(* PLC project mtcs, Institute of Astronomy OntoManager 0.0.1 *)
(* stored: creationDateTime 2017-02-07T02:01:16.949163, modificationDateTime 2017-02-07T02:01:16.949163 *)

TYPE MTCSParts : STRUCT
  telemetry : Telemetry;  (* The telemetry *)
  cover : Cover;  (* The Cover of the telescope *)
  m1 : M1;  (* The primary mirror of the telescope *)
  m2 : M2;  (* The secondary mirror of the telescope *)
  m3 : M3;  (* The tertiary mirror of the telescope *)
  services : Services;  (* The Services system *)
  safety : Safety;  (* The safety *)
  hydraulics : Hydraulics;  (* The hydraulics *)
  axes : Axes;  (* The axes *)
  dome : Dome;  (* The dome *)
  configManager : ConfigManager;  (* The config manager (to load/save/activate configuration data) *)
END_STRUCT;
END_TYPE

TYPE MTCSProcesses : STRUCT
  initialize : Process;  (* Start initializing the whole MTCS *)
  lock : Process;  (* Lock the whole MTCS *)
  unlock : Process;  (* Unlock the whole MTCS *)
  changeOperator : ChangeOperatorStateProcess;  (* Change the operator (e.g. OBSERVER, TECH, ...) *)
  verifyPassword : ChangeOperatorStateProcess;  (* Only verify the operator password *)
  reboot : Process;  (* Reboot the whole MTCS *)
  shutdown : Process;  (* Shutdown the whole MTCS *)
  wakeUp : Process;  (* Wake up the whole MTCS *)
  goToSleep : Process;  (* Let the whole MTCS go to sleep *)
  stop : Process;  (* Stop the dome and telescope *)
  endOfNight : Process;  (* End of night *)
  changeInstrument : MTCSChangeInstrumentProcess;  (* Change the instrument *)
  park : MTCSParkProcess;  (* Park the telescope (including Axes, Dome, M3, ...) *)
  point : MTCSPointProcess;  (* Point the telescope and dome to a new target *)
END_STRUCT;
END_TYPE

TYPE MTCSStatuses : STRUCT
  initializationStatus : InitializationStatus;
  healthStatus : HealthStatus;
  busyStatus : BusyStatus;
  operatorStatus : OperatorStatus;
  passwordHealthStatus : HealthStatus;
  activityStatus : ActivityStatus;
END_STRUCT;
END_TYPE

TYPE MTCSInstrumentsConfig : STRUCT
  instrument0 : InstrumentConfig;  (* Instrument 0 *)
  instrument1 : InstrumentConfig;  (* Instrument 1 *)
  instrument2 : InstrumentConfig;  (* Instrument 2 *)
  instrument3 : InstrumentConfig;  (* Instrument 3 *)
  instrument4 : InstrumentConfig;  (* Instrument 4 *)
  instrument5 : InstrumentConfig;  (* Instrument 5 *)
  instrument6 : InstrumentConfig;  (* Instrument 6 *)
  instrument7 : InstrumentConfig;  (* Instrument 7 *)
  instrument8 : InstrumentConfig;  (* Instrument 8 *)
  instrument9 : InstrumentConfig;  (* Instrument 9 *)
END_STRUCT;
END_TYPE

TYPE MTCSParkPositionConfig : STRUCT
  name : STRING;  (* The name of the position (e.g. 'PARK') *)
  axes : STRING;  (* Name of the corresponding Axes position *)
  doAxes : BOOL;  (* Change the Axes to the 'axes' position *)
  m3 : STRING;  (* Name of the corresponding M3 position *)
  doM3 : BOOL;  (* Change M3 to the 'm3' position *)
  dome : STRING;  (* Name of the corresponding dome position *)
  doDome : BOOL;  (* Change M3 to the 'm3' position *)
END_STRUCT;
END_TYPE

TYPE MTCSParkPositionsConfig : STRUCT
  position0 : MTCSParkPositionConfig;  (* Park position 0 *)
  position1 : MTCSParkPositionConfig;  (* Park position 1 *)
  position2 : MTCSParkPositionConfig;  (* Park position 2 *)
  position3 : MTCSParkPositionConfig;  (* Park position 3 *)
  position4 : MTCSParkPositionConfig;  (* Park position 4 *)
  position5 : MTCSParkPositionConfig;  (* Park position 5 *)
  position6 : MTCSParkPositionConfig;  (* Park position 6 *)
  position7 : MTCSParkPositionConfig;  (* Park position 7 *)
  position8 : MTCSParkPositionConfig;  (* Park position 8 *)
  position9 : MTCSParkPositionConfig;  (* Park position 9 *)
END_STRUCT;
END_TYPE

TYPE MTCSEndOfNightStepConfig : STRUCT
  parkAxes : BOOL;  (* Park the telescope *)
  parkAxesPosition : STRING;  (* Position to park the telescope *)
  parkTelescopeWait : BOOL;  (* Wait until the telescope is parked *)
  parkM3 : BOOL;  (* Park M3 *)
  parkM3Position : STRING;  (* Position to park M3 *)
  parkM3Wait : BOOL;  (* Wait until M3 is parked *)
  parkDome : BOOL;  (* Park the dome *)
  parkDomePosition : STRING;  (* Position to park the dome *)
  parkDomeWait : BOOL;  (* Wait until the dome is parked *)
  closeCover : BOOL;  (* Close the cover *)
  closeCoverWait : BOOL;  (* Wait until the cover is closed *)
  closeDome : BOOL;  (* Close the dome *)
  closeDomeWait : BOOL;  (* Wait until the dome is closed *)
  stop : BOOL;  (* Stop the axes and dome *)
  stopWait : BOOL;  (* Wait until the axes and dome are stopped *)
  goToSleep : BOOL;  (* Make the telescope go to sleep *)
  goToSleepWait : BOOL;  (* Wait until the telescope is sleeping *)
END_STRUCT;
END_TYPE

TYPE MTCSEndOfNightConfig : STRUCT
  step0 : MTCSEndOfNightStepConfig;  (* Step 0 *)
  step1 : MTCSEndOfNightStepConfig;  (* Step 1 *)
  step2 : MTCSEndOfNightStepConfig;  (* Step 2 *)
  step3 : MTCSEndOfNightStepConfig;  (* Step 3 *)
  step4 : MTCSEndOfNightStepConfig;  (* Step 4 *)
  step5 : MTCSEndOfNightStepConfig;  (* Step 5 *)
  step6 : MTCSEndOfNightStepConfig;  (* Step 6 *)
  step7 : MTCSEndOfNightStepConfig;  (* Step 7 *)
  step8 : MTCSEndOfNightStepConfig;  (* Step 8 *)
  step9 : MTCSEndOfNightStepConfig;  (* Step 9 *)
  step10 : MTCSEndOfNightStepConfig;  (* Step 10 *)
  step11 : MTCSEndOfNightStepConfig;  (* Step 11 *)
  step12 : MTCSEndOfNightStepConfig;  (* Step 12 *)
  step13 : MTCSEndOfNightStepConfig;  (* Step 13 *)
  step14 : MTCSEndOfNightStepConfig;  (* Step 14 *)
  step15 : MTCSEndOfNightStepConfig;  (* Step 15 *)
  step16 : MTCSEndOfNightStepConfig;  (* Step 16 *)
  step17 : MTCSEndOfNightStepConfig;  (* Step 17 *)
  step18 : MTCSEndOfNightStepConfig;  (* Step 18 *)
  step19 : MTCSEndOfNightStepConfig;  (* Step 19 *)
END_STRUCT;
END_TYPE

TYPE MTCSConfig : STRUCT
  instruments : MTCSInstrumentsConfig;  (* Configure the instruments *)
  endOfNight : MTCSEndOfNightConfig;  (* Configure the instruments *)
  parkPositions : MTCSParkPositionsConfig;  (* Configure the park positions of the telescope (dome+telescope+m3+...) *)
END_STRUCT;
END_TYPE

TYPE MTCSChangeInstrumentProcessArgs : STRUCT
  name : STRING;  (* Name of the instrument *)
END_STRUCT;
END_TYPE

TYPE MTCSParkProcessArgs : STRUCT
  name : STRING;  (* Name of the park position *)
END_STRUCT;
END_TYPE

TYPE MTCSPointProcessArgs : STRUCT
  alphaUnits : AxesAlphaUnits;  (* The units in which alpha is given *)
  alpha : LREAL;  (* Right ascention, in the units of the alphaUnits argument *)
  deltaUnits : AxesDeltaUnits;  (* The units in which delta is given *)
  delta : LREAL;  (* Declination, in the units of the deltaUnits argument *)
  muUnits : AxesMuUnits;  (* The units in which muAlpha and muDelta are given *)
  muAlpha : LREAL;  (* Right ascention proper motion, the units of muUmits (do not multiply by cos(delta)!) *)
  muDelta : LREAL;  (* Declination proper motion, in radians/year *)
  parallax : LREAL;  (* Object parallax, in arcseconds *)
  radialVelocity : LREAL;  (* Object radial velocity, in km/s *)
  epoch : LREAL := 2000;  (* Epoch, e.g. 2000.0 *)
  tracking : BOOL := TRUE;  (* True to start tracking the object, false to Only do a pointing *)
  rotUnits : AxesMoveUnits;  (* Units of the 'rot', 'roc' and 'ron' arguments (RADIANS, DEGREES, ARCSECONDS, ...) *)
  rotOffset : LREAL;  (* Offset to move the currently active rotator (incompatible with 'roc' and 'ron' args) *)
  rocOffset : LREAL;  (* Offset to move the cassegrain rotation axis (incompatible with 'rot' arg) *)
  ronOffset : LREAL;  (* Offset to move the nasmyth rotation axis (incompatible with 'rot' arg) *)
  doRotOffset : BOOL;  (* True to move the currently active rotator, false to leave it untouched *)
  doRocOffset : BOOL;  (* True to move the cassegrain rotation axis, false to leave it untouched *)
  doRonOffset : BOOL;  (* True to move the nasmyth rotation axis, false to leave it untouched *)
  doDomeTracking : BOOL := TRUE;  (* True to enable dome tracking *)
END_STRUCT;
END_TYPE

FUNCTION_BLOCK SM_MTCS
  VAR_INPUT
    {attribute 'OPC.UA.DA' := '1'}
    {attribute 'OPC.UA.DA.Access' := '1'}
    editableConfig : MTCSConfig;  (* Editable configuration of the MTCS *)
  END_VAR
  VAR_OUTPUT
    {attribute 'OPC.UA.DA' := '1'}
    {attribute 'OPC.UA.DA.Access' := '1'}
    actualStatus : STRING;  (* Current status description *)
    previousStatus : STRING;  (* Previous status description *)
    {attribute 'OPC.UA.DA' := '1'}
    {attribute 'OPC.UA.DA.Access' := '1'}
    noOfFailedOperatorChanges : UINT;  (* How many times has a wrong password been entered? *)
    {attribute 'OPC.UA.DA' := '1'}
    {attribute 'OPC.UA.DA.Access' := '1'}
    activeInstrument : InstrumentConfig;  (* Config of the currently active instrument (depending on M3 and possibly derotator) *if* isInstrumentActive is TRUE *)
    {attribute 'OPC.UA.DA' := '1'}
    {attribute 'OPC.UA.DA.Access' := '1'}
    activeInstrumentNumber : INT;  (* Number of the currently active instrument (0..9, or -1 if no instrument is active) *)
    {attribute 'OPC.UA.DA' := '1'}
    {attribute 'OPC.UA.DA.Access' := '1'}
    activeInstrumentName : STRING;  (* Name of the currently active instrument *)
    {attribute 'OPC.UA.DA' := '1'}
    {attribute 'OPC.UA.DA.Access' := '1'}
    isInstrumentActive : BOOL;  (* Is an instrument currently active (i.e. is M3 static at a known position?) *)
    {attribute 'OPC.UA.DA' := '1'}
    {attribute 'OPC.UA.DA.Access' := '1'}
    config : MTCSConfig;  (* Active configuration of the ServicesTiming subsystem *)
    statuses : MTCSStatuses;  (* Statuses of the state machine *)
    parts : MTCSParts;  (* Parts of the state machine *)
    processes : MTCSProcesses;  (* Processes of the state machine *)
  END_VAR

            parts.telemetry( operatorStatus := statuses.operatorStatus );
parts.cover(
    operatorStatus := statuses.operatorStatus,
    aziPos := parts.axes.parts.azi.actPos,
    elePos := parts.axes.parts.ele.actPos);
parts.m1(
    operatorStatus := statuses.operatorStatus,
    tubeAngleMeasurement := parts.telemetry.parts.accelerometers.tube);
parts.m2(
    operatorStatus := statuses.operatorStatus,
    io := parts.m1.parts.io,
    actualFocalStation := parts.m3.actualKnownPositionID,
    m3KnownPositionsConfig := parts.m3.config.knownPositions,
    temperatures := parts.telemetry.parts.temperatures);
parts.m3( operatorStatus := statuses.operatorStatus );
parts.services( operatorStatus := statuses.operatorStatus );
parts.safety(
    operatorStatus := statuses.operatorStatus,
    activityStatus := statuses.activityStatus);
parts.hydraulics(
    operatorStatus := statuses.operatorStatus,
    safetyHydraulics := parts.safety.parts.hydraulics,
    safetyIO := parts.safety.parts.io);
parts.dome(
    operatorStatus := statuses.operatorStatus,
    aziPos := parts.axes.parts.azi.actPos);
parts.configManager( isEnabled := statuses.operatorStatus.tech );
statuses.initializationStatus();
statuses.healthStatus(
    isGood := parts.axes.statuses.healthStatus.isGood AND (parts.cover.statuses.healthStatus.isGood AND (parts.m1.statuses.healthStatus.isGood AND (parts.m2.statuses.healthStatus.isGood AND (parts.m3.statuses.healthStatus.isGood AND (parts.services.statuses.healthStatus.isGood AND (parts.telemetry.statuses.healthStatus.isGood AND (parts.safety.statuses.healthStatus.isGood AND (parts.hydraulics.statuses.healthStatus.isGood AND parts.dome.statuses.healthStatus.isGood)))))))),
    hasWarning := parts.axes.statuses.healthStatus.hasWarning OR (parts.cover.statuses.healthStatus.hasWarning OR (parts.m1.statuses.healthStatus.hasWarning OR (parts.m2.statuses.healthStatus.hasWarning OR (parts.m3.statuses.healthStatus.hasWarning OR (parts.services.statuses.healthStatus.hasWarning OR (parts.telemetry.statuses.healthStatus.hasWarning OR (parts.safety.statuses.healthStatus.hasWarning OR (parts.hydraulics.statuses.healthStatus.hasWarning OR parts.dome.statuses.healthStatus.hasWarning)))))))));
statuses.busyStatus( isBusy := parts.axes.statuses.busyStatus.busy OR (parts.cover.statuses.busyStatus.busy OR (parts.m1.statuses.busyStatus.busy OR (parts.m2.statuses.busyStatus.busy OR (parts.m3.statuses.busyStatus.busy OR (parts.services.statuses.busyStatus.busy OR (parts.telemetry.statuses.busyStatus.busy OR (parts.safety.statuses.busyStatus.busy OR (parts.hydraulics.statuses.busyStatus.busy OR parts.dome.statuses.busyStatus.busy)))))))) );
statuses.operatorStatus();
statuses.passwordHealthStatus( superState := statuses.operatorStatus.observer );
statuses.activityStatus(
    superState := statuses.initializationStatus.initialized OR statuses.initializationStatus.initializingFailed,
    isAwake := (parts.hydraulics.pumpsState = HydraulicsPumpsStates.RUNNING) OR parts.axes.statuses.poweredStatus.enabled,
    isMoving := parts.axes.statuses.busyStatus.busy OR parts.axes.isTracking);
processes.initialize( isEnabled := NOT(statuses.initializationStatus.initializing) );
processes.lock( isEnabled := statuses.operatorStatus.tech AND statuses.initializationStatus.initialized );
processes.unlock( isEnabled := statuses.operatorStatus.tech AND statuses.initializationStatus.locked );
processes.changeOperator( isEnabled := TRUE );
processes.verifyPassword( isEnabled := TRUE );
processes.reboot( isEnabled := TRUE );
processes.shutdown( isEnabled := statuses.operatorStatus.tech );
processes.wakeUp( isEnabled := statuses.activityStatus.sleeping );
processes.goToSleep( isEnabled := statuses.activityStatus.awake OR statuses.healthStatus.bad );
processes.stop( isEnabled := statuses.initializationStatus.initialized );
processes.endOfNight( isEnabled := TRUE );
processes.changeInstrument( isEnabled := statuses.initializationStatus.initialized OR statuses.healthStatus.bad );
processes.park( isEnabled := parts.axes.statuses.busyStatus.idle AND (parts.dome.statuses.busyStatus.idle AND parts.m3.statuses.busyStatus.idle) );
processes.point( isEnabled := parts.axes.processes.point.statuses.enabledStatus.enabled AND parts.dome.processes.trackAxes.statuses.enabledStatus.enabled );

          

{attribute 'TcRpcEnable' := '1'}
METHOD initialize : RequestResults
                  initialize := THIS^.processes.initialize.request();

                
END_METHOD

{attribute 'TcRpcEnable' := '1'}
METHOD lock : RequestResults
                  lock := THIS^.processes.lock.request();

                
END_METHOD

{attribute 'TcRpcEnable' := '1'}
METHOD unlock : RequestResults
                  unlock := THIS^.processes.unlock.request();

                
END_METHOD

{attribute 'TcRpcEnable' := '1'}
METHOD changeOperator : RequestResults
  VAR_INPUT
    state : OperatorStates;
    password : STRING;
  END_VAR
                  changeOperator := THIS^.processes.changeOperator.request(
    state := state,
    password := password);

                
END_METHOD

{attribute 'TcRpcEnable' := '1'}
METHOD verifyPassword : RequestResults
  VAR_INPUT
    state : OperatorStates;
    password : STRING;
  END_VAR
                  verifyPassword := THIS^.processes.verifyPassword.request(
    state := state,
    password := password);

                
END_METHOD

{attribute 'TcRpcEnable' := '1'}
METHOD reboot : RequestResults
                  reboot := THIS^.processes.reboot.request();

                
END_METHOD

{attribute 'TcRpcEnable' := '1'}
METHOD shutdown : RequestResults
                  shutdown := THIS^.processes.shutdown.request();

                
END_METHOD

{attribute 'TcRpcEnable' := '1'}
METHOD wakeUp : RequestResults
                  wakeUp := THIS^.processes.wakeUp.request();

                
END_METHOD

{attribute 'TcRpcEnable' := '1'}
METHOD goToSleep : RequestResults
                  goToSleep := THIS^.processes.goToSleep.request();

                
END_METHOD

{attribute 'TcRpcEnable' := '1'}
METHOD stop : RequestResults
                  stop := THIS^.processes.stop.request();

                
END_METHOD

{attribute 'TcRpcEnable' := '1'}
METHOD endOfNight : RequestResults
                  endOfNight := THIS^.processes.endOfNight.request();

                
END_METHOD

{attribute 'TcRpcEnable' := '1'}
METHOD changeInstrument : RequestResults
  VAR_INPUT
    name : STRING;
  END_VAR
                  changeInstrument := THIS^.processes.changeInstrument.request( name := name );

                
END_METHOD

{attribute 'TcRpcEnable' := '1'}
METHOD park : RequestResults
  VAR_INPUT
    name : STRING;
  END_VAR
                  park := THIS^.processes.park.request( name := name );

                
END_METHOD

{attribute 'TcRpcEnable' := '1'}
METHOD point : RequestResults
  VAR_INPUT
    alphaUnits : AxesAlphaUnits;
    alpha : LREAL;
    deltaUnits : AxesDeltaUnits;
    delta : LREAL;
    muUnits : AxesMuUnits;
    muAlpha : LREAL;
    muDelta : LREAL;
    parallax : LREAL;
    radialVelocity : LREAL;
    epoch : LREAL;
    tracking : BOOL;
    rotUnits : AxesMoveUnits;
    rotOffset : LREAL;
    rocOffset : LREAL;
    ronOffset : LREAL;
    doRotOffset : BOOL;
    doRocOffset : BOOL;
    doRonOffset : BOOL;
    doDomeTracking : BOOL;
  END_VAR
                  point := THIS^.processes.point.request(
    alphaUnits := alphaUnits,
    alpha := alpha,
    deltaUnits := deltaUnits,
    delta := delta,
    muUnits := muUnits,
    muAlpha := muAlpha,
    muDelta := muDelta,
    parallax := parallax,
    radialVelocity := radialVelocity,
    epoch := epoch,
    tracking := tracking,
    rotUnits := rotUnits,
    rotOffset := rotOffset,
    rocOffset := rocOffset,
    ronOffset := ronOffset,
    doRotOffset := doRotOffset,
    doRocOffset := doRocOffset,
    doRonOffset := doRonOffset,
    doDomeTracking := doDomeTracking);

                
END_METHOD

{attribute 'TcRpcEnable' := '1'}
METHOD _log : BOOL
  VAR_INPUT
    name : STRING;  (* Name of this function block instance *)
  END_VAR
  VAR_IN_OUT
    buffer : LogBuffer;  (* Buffer to write all logging to *)
  END_VAR
  VAR
    subBuffer : LogBuffer;  (* Temporary buffer to write logging by parts (sub-statemachines) to *)
  END_VAR
                  THIS^.parts.telemetry._log(
    name := 'telemetry',
    buffer := subBuffer);
THIS^.parts.cover._log(
    name := 'cover',
    buffer := subBuffer);
THIS^.parts.m1._log(
    name := 'm1',
    buffer := subBuffer);
THIS^.parts.m2._log(
    name := 'm2',
    buffer := subBuffer);
THIS^.parts.m3._log(
    name := 'm3',
    buffer := subBuffer);
THIS^.parts.services._log(
    name := 'services',
    buffer := subBuffer);
THIS^.parts.safety._log(
    name := 'safety',
    buffer := subBuffer);
THIS^.parts.hydraulics._log(
    name := 'hydraulics',
    buffer := subBuffer);
THIS^.parts.axes._log(
    name := 'axes',
    buffer := subBuffer);
THIS^.parts.dome._log(
    name := 'dome',
    buffer := subBuffer);
THIS^.parts.configManager._log(
    name := 'configManager',
    buffer := subBuffer);
LOGGER(
    name := name,
    actualStatus := THIS^.actualStatus,
    previousStatus := THIS^.previousStatus,
    buffer := buffer,
    subBuffer := subBuffer,
    pHealthStatus := ADR(THIS^.statuses.healthStatus),
    pBusyStatus := ADR(THIS^.statuses.busyStatus));

                
END_METHOD
END_FUNCTION_BLOCK

FUNCTION_BLOCK MTCSChangeInstrumentProcess EXTENDS BaseProcess
  VAR_INPUT
    {attribute 'OPC.UA.DA' := '1'}
    set : MTCSChangeInstrumentProcessArgs;  (* Arguments to be set, before writing do_request TRUE *)
  END_VAR
  VAR_OUTPUT
    {attribute 'OPC.UA.DA' := '1'}
    {attribute 'OPC.UA.DA.Access' := '1'}
    get : MTCSChangeInstrumentProcessArgs;  (* Arguments in use by the process, if do_request was accepted *)
  END_VAR

            IF do_request THEN
    do_request_result := request( name := set.name );
    do_request := FALSE;
END_IF;
SUPER^();

          

{attribute 'TcRpcEnable' := '1'}
METHOD start
  VAR_INPUT
    name : STRING;  (* Name of the instrument *)
  END_VAR
                  THIS^.get.name := name;
THIS^.statuses.busyStatus( isBusy := TRUE );
THIS^.statuses.healthStatus( isGood := TRUE );

                
END_METHOD

{attribute 'TcRpcEnable' := '1'}
METHOD request : RequestResults
  VAR_INPUT
    name : STRING;  (* Name of the instrument *)
  END_VAR
                  IF THIS^.statuses.enabledStatus.enabled THEN
    THIS^.start( name := name );
    request := RequestResults.ACCEPTED;
ELSE
    request := RequestResults.REJECTED;
END_IF;

                
END_METHOD
END_FUNCTION_BLOCK

FUNCTION_BLOCK MTCSParkProcess EXTENDS BaseProcess
  VAR_INPUT
    {attribute 'OPC.UA.DA' := '1'}
    set : MTCSParkProcessArgs;  (* Arguments to be set, before writing do_request TRUE *)
  END_VAR
  VAR_OUTPUT
    {attribute 'OPC.UA.DA' := '1'}
    {attribute 'OPC.UA.DA.Access' := '1'}
    get : MTCSParkProcessArgs;  (* Arguments in use by the process, if do_request was accepted *)
  END_VAR

            IF do_request THEN
    do_request_result := request( name := set.name );
    do_request := FALSE;
END_IF;
SUPER^();

          

{attribute 'TcRpcEnable' := '1'}
METHOD start
  VAR_INPUT
    name : STRING;  (* Name of the park position *)
  END_VAR
                  THIS^.get.name := name;
THIS^.statuses.busyStatus( isBusy := TRUE );
THIS^.statuses.healthStatus( isGood := TRUE );

                
END_METHOD

{attribute 'TcRpcEnable' := '1'}
METHOD request : RequestResults
  VAR_INPUT
    name : STRING;  (* Name of the park position *)
  END_VAR
                  IF THIS^.statuses.enabledStatus.enabled THEN
    THIS^.start( name := name );
    request := RequestResults.ACCEPTED;
ELSE
    request := RequestResults.REJECTED;
END_IF;

                
END_METHOD
END_FUNCTION_BLOCK

FUNCTION_BLOCK MTCSPointProcess EXTENDS BaseProcess
  VAR_INPUT
    {attribute 'OPC.UA.DA' := '1'}
    set : MTCSPointProcessArgs;  (* Arguments to be set, before writing do_request TRUE *)
  END_VAR
  VAR_OUTPUT
    {attribute 'OPC.UA.DA' := '1'}
    {attribute 'OPC.UA.DA.Access' := '1'}
    get : MTCSPointProcessArgs;  (* Arguments in use by the process, if do_request was accepted *)
  END_VAR

            IF do_request THEN
    do_request_result := request(
    alphaUnits := set.alphaUnits,
    alpha := set.alpha,
    deltaUnits := set.deltaUnits,
    delta := set.delta,
    muUnits := set.muUnits,
    muAlpha := set.muAlpha,
    muDelta := set.muDelta,
    parallax := set.parallax,
    radialVelocity := set.radialVelocity,
    epoch := set.epoch,
    tracking := set.tracking,
    rotUnits := set.rotUnits,
    rotOffset := set.rotOffset,
    rocOffset := set.rocOffset,
    ronOffset := set.ronOffset,
    doRotOffset := set.doRotOffset,
    doRocOffset := set.doRocOffset,
    doRonOffset := set.doRonOffset,
    doDomeTracking := set.doDomeTracking);
    do_request := FALSE;
END_IF;
SUPER^();

          

{attribute 'TcRpcEnable' := '1'}
METHOD start
  VAR_INPUT
    alphaUnits : AxesAlphaUnits;  (* The units in which alpha is given *)
    alpha : LREAL;  (* Right ascention, in the units of the alphaUnits argument *)
    deltaUnits : AxesDeltaUnits;  (* The units in which delta is given *)
    delta : LREAL;  (* Declination, in the units of the deltaUnits argument *)
    muUnits : AxesMuUnits;  (* The units in which muAlpha and muDelta are given *)
    muAlpha : LREAL;  (* Right ascention proper motion, the units of muUmits (do not multiply by cos(delta)!) *)
    muDelta : LREAL;  (* Declination proper motion, in radians/year *)
    parallax : LREAL;  (* Object parallax, in arcseconds *)
    radialVelocity : LREAL;  (* Object radial velocity, in km/s *)
    epoch : LREAL := 2000;  (* Epoch, e.g. 2000.0 *)
    tracking : BOOL := TRUE;  (* True to start tracking the object, false to Only do a pointing *)
    rotUnits : AxesMoveUnits;  (* Units of the 'rot', 'roc' and 'ron' arguments (RADIANS, DEGREES, ARCSECONDS, ...) *)
    rotOffset : LREAL;  (* Offset to move the currently active rotator (incompatible with 'roc' and 'ron' args) *)
    rocOffset : LREAL;  (* Offset to move the cassegrain rotation axis (incompatible with 'rot' arg) *)
    ronOffset : LREAL;  (* Offset to move the nasmyth rotation axis (incompatible with 'rot' arg) *)
    doRotOffset : BOOL;  (* True to move the currently active rotator, false to leave it untouched *)
    doRocOffset : BOOL;  (* True to move the cassegrain rotation axis, false to leave it untouched *)
    doRonOffset : BOOL;  (* True to move the nasmyth rotation axis, false to leave it untouched *)
    doDomeTracking : BOOL := TRUE;  (* True to enable dome tracking *)
  END_VAR
                  THIS^.get.alphaUnits := alphaUnits;
THIS^.get.alpha := alpha;
THIS^.get.deltaUnits := deltaUnits;
THIS^.get.delta := delta;
THIS^.get.muUnits := muUnits;
THIS^.get.muAlpha := muAlpha;
THIS^.get.muDelta := muDelta;
THIS^.get.parallax := parallax;
THIS^.get.radialVelocity := radialVelocity;
THIS^.get.epoch := epoch;
THIS^.get.tracking := tracking;
THIS^.get.rotUnits := rotUnits;
THIS^.get.rotOffset := rotOffset;
THIS^.get.rocOffset := rocOffset;
THIS^.get.ronOffset := ronOffset;
THIS^.get.doRotOffset := doRotOffset;
THIS^.get.doRocOffset := doRocOffset;
THIS^.get.doRonOffset := doRonOffset;
THIS^.get.doDomeTracking := doDomeTracking;
THIS^.statuses.busyStatus( isBusy := TRUE );
THIS^.statuses.healthStatus( isGood := TRUE );

                
END_METHOD

{attribute 'TcRpcEnable' := '1'}
METHOD request : RequestResults
  VAR_INPUT
    alphaUnits : AxesAlphaUnits;  (* The units in which alpha is given *)
    alpha : LREAL;  (* Right ascention, in the units of the alphaUnits argument *)
    deltaUnits : AxesDeltaUnits;  (* The units in which delta is given *)
    delta : LREAL;  (* Declination, in the units of the deltaUnits argument *)
    muUnits : AxesMuUnits;  (* The units in which muAlpha and muDelta are given *)
    muAlpha : LREAL;  (* Right ascention proper motion, the units of muUmits (do not multiply by cos(delta)!) *)
    muDelta : LREAL;  (* Declination proper motion, in radians/year *)
    parallax : LREAL;  (* Object parallax, in arcseconds *)
    radialVelocity : LREAL;  (* Object radial velocity, in km/s *)
    epoch : LREAL := 2000;  (* Epoch, e.g. 2000.0 *)
    tracking : BOOL := TRUE;  (* True to start tracking the object, false to Only do a pointing *)
    rotUnits : AxesMoveUnits;  (* Units of the 'rot', 'roc' and 'ron' arguments (RADIANS, DEGREES, ARCSECONDS, ...) *)
    rotOffset : LREAL;  (* Offset to move the currently active rotator (incompatible with 'roc' and 'ron' args) *)
    rocOffset : LREAL;  (* Offset to move the cassegrain rotation axis (incompatible with 'rot' arg) *)
    ronOffset : LREAL;  (* Offset to move the nasmyth rotation axis (incompatible with 'rot' arg) *)
    doRotOffset : BOOL;  (* True to move the currently active rotator, false to leave it untouched *)
    doRocOffset : BOOL;  (* True to move the cassegrain rotation axis, false to leave it untouched *)
    doRonOffset : BOOL;  (* True to move the nasmyth rotation axis, false to leave it untouched *)
    doDomeTracking : BOOL := TRUE;  (* True to enable dome tracking *)
  END_VAR
                  IF THIS^.statuses.enabledStatus.enabled THEN
    THIS^.start(
        alphaUnits := alphaUnits,
        alpha := alpha,
        deltaUnits := deltaUnits,
        delta := delta,
        muUnits := muUnits,
        muAlpha := muAlpha,
        muDelta := muDelta,
        parallax := parallax,
        radialVelocity := radialVelocity,
        epoch := epoch,
        tracking := tracking,
        rotUnits := rotUnits,
        rotOffset := rotOffset,
        rocOffset := rocOffset,
        ronOffset := ronOffset,
        doRotOffset := doRotOffset,
        doRocOffset := doRocOffset,
        doRonOffset := doRonOffset,
        doDomeTracking := doDomeTracking);
    request := RequestResults.ACCEPTED;
ELSE
    request := RequestResults.REJECTED;
END_IF;

                
END_METHOD
END_FUNCTION_BLOCK
